FUNCTION_BLOCK FB_FrameFifo_2
VAR_INPUT
	bLog		: BOOL := FALSE;
	stPut		: ST_FrameFifoEntrydata_2;
	
END_VAR
VAR_OUTPUT
	bOk			: BOOL;
	stGet		: ST_FrameFifoEntrydata_2;
	nCount		: UDINT := 0;
END_VAR
VAR
	fbBuffer 	: FB_MemRingBuffer;
	buffer		: ARRAY[0..NUMBER_OF_BYTE_FOR_ALL_FRAMEFIFO] OF BYTE;
	i : INT;
END_VAR
VAR CONSTANT
	SIZE_OF_FRAMEFIFO : UDINT := SIZEOF(ST_FrameFifoEntrydata_2);
	MAX_NUMBER_OF_FRAMEFIFO : UDINT := 10;
	NUMBER_OF_BYTE_FOR_ALL_FRAMEFIFO : UDINT := SIZE_OF_FRAMEFIFO*MAX_NUMBER_OF_FRAMEFIFO;
END_VAR

;

ACTION AddTail:

fbBuffer.A_AddTail( pBuffer:= ADR(buffer), cbBuffer:= SIZEOF(buffer),
					pWrite:= ADR( stPut ), cbWrite := SIZEOF( stPut ), 
					bOk=>bOk, nCount=>nCount );
END_ACTION

ACTION Clear:

FOR i:=0 TO TXDATASIZE_2 BY 1 DO
stget.txdata[i] := 0;
END_FOR


stGet.stRemoteAddr.nPort := 0;
stGet.stRemoteAddr.sAddr := '';
fbBuffer.A_Reset( pBuffer := ADR( buffer ), cbBuffer := SIZEOF( buffer ), 
					bOk=>bOk, nCount=>nCount );
END_ACTION

ACTION RemoveHead:

IF nCount = 0 THEN	 

FOR i:=0 TO TXDATASIZE_2 BY 1 DO
stget.txdata[i] := 0;
END_FOR
	stGet.stRemoteAddr.nPort := 0;
	stGet.stRemoteAddr.sAddr := '';
	bOk := FALSE;
	RETURN;
END_IF

fbBuffer.A_RemoveHead( pBuffer:= ADR(buffer), cbBuffer:= SIZEOF(buffer),
						pRead := ADR( stGet ), cbRead := SIZEOF( stGet ),
						bOk=>bOk, nCount=>nCount );
END_ACTION

END_FUNCTION_BLOCK

(* stored: Version 1.1.0.1, ProductVersion 3.1.4024.13
   POU FB_FrameFifo_2: Id {726adbbc-8593-42b1-a82a-01b4716d9adb}, SpecialFunc None
   Action AddTail: Id {cd34f04f-c317-4bf9-8dee-ada79687db57}
   Action Clear: Id {59f6a1b0-697c-415c-92e7-db31c6829484}
   Action RemoveHead: Id {6af1ed2c-86f4-4919-992b-aeaf42f0b210} *)
